// TIA Portal V17 export
// export: Created 2024-09-03T21:54:52.8265219Z, ExportSetting WithDefaults, DisplayName Totally Integrated Automation Portal, DisplayVersion V17 Update 7, DisplayName TIA Portal Openness, DisplayVersion V17 Update 7, DisplayName TIA Portal Version Control Interface, DisplayVersion V17, DisplayName SINAMICS Startdrive Advanced, DisplayVersion V17 SP2, DisplayName SINAMICS Startdrive G110M, G120, G120C, G120D, G120P, G115D, DisplayVersion V17 SP2, DisplayName SINAMICS Startdrive G130, G150, S120, S150, SINAMICS MV, S210, DisplayVersion V17 SP2, DisplayName STEP 7 Professional, DisplayVersion V17 Update 7, DisplayName STEP 7 Safety, DisplayVersion V17 Update 6, DisplayName WinCC Advanced / Unified PC, DisplayVersion V17 Update 7
FUNCTION_BLOCK "FB_Eks"   // FB5050, LAD
{ S7_Optimized_Access := 'TRUE' }
VERSION : 0.1
// stored: AutoNumber false, IsIECCheckEnabled false, IsRetainMemResEnabled false, MemoryReserve 100, SetENOAutomatically false, UDAEnableTagReadback false
   VAR_INPUT
      iScreenNumberEqual : Bool;
      iOpSwitchManualMode : Bool;
      iGenerateTimeoutError : Bool;
      iPermanentAccess : Bool;
      iBlinker : Bool;
   END_VAR
   VAR_OUTPUT
      qManualModeActive : Bool;
      qOpManualModeLamp : Bool;
      qeKeyTimeout : Bool;
   END_VAR
   VAR DB_SPECIFIC
      Status : Struct
         Key : Struct
            Inserted : Bool;
            Found : Bool;
            Valid : Bool;
            ActualKeyStatus : Int;   // 0= Not inserted, ??= GAP leader, ??= Maintenance, ??= Engineer, 100= Not registered
            LastKeyStatus : Int;   // 0= Not used, ??= GAP leader, ??= Maintenance, ??= Engineer, 100= Not registered
         END_STRUCT;
         Global : Struct
            GapLeader : Bool;
            Maintenance : Bool;
            Engineer : Bool;
            MaintenanceOrEngineer : Bool;
            AnyValidKey : Bool;
         END_STRUCT;
         ManualMode : Struct
            GapLeader : Bool;
            Maintenance : Bool;
            Engineer : Bool;
            MaintenanceOrEngineer : Bool;
            AnyValidKey : Bool;
         END_STRUCT;
      END_STRUCT;
   END_VAR
   VAR
      Database : Struct
         Status : Struct
            ActualAndLastKeyEqual { ExternalAccessible := 'False'; ExternalVisible := 'False'; ExternalWritable := 'False'} : Bool;
            LastKeyIsEmpty : Bool;
            LastKeyEmployeeIDIsEmpty : Bool;
            LastKeyFound { ExternalAccessible := 'False'; ExternalVisible := 'False'; ExternalWritable := 'False'} : Bool;
            LastKeyIndex { ExternalAccessible := 'False'; ExternalVisible := 'False'; ExternalWritable := 'False'} : Int;
            FreePlaceFound { ExternalAccessible := 'False'; ExternalVisible := 'False'; ExternalWritable := 'False'} : Bool;
            FreePlaceIndex { ExternalAccessible := 'False'; ExternalVisible := 'False'; ExternalWritable := 'False'} : Int;
            NumberOfKeys : Int;
            NumberOfStoredKeys : Int;
            StoredKeysReachedMaximum : Bool;
            NumberOfEngineerKeys : Int;
            NumberOfStoredEngineerKeys : Int;
            StoredEngineerKeysReachedMaximum : Bool;
         END_STRUCT;
         ListNumber : Int;
         ListNumberLast : Int;
      END_STRUCT;
   END_VAR
   VAR DB_SPECIFIC
      KeyManage : Struct
         CanBeAdd : Bool;
         Add : Bool;
         CanBeRemoved : Bool;
         Remove : Bool;
         CanBeUsed : Bool;
         Use : Int;
         CanBeSearched : Bool;
         Search : Bool;
         Searching : Bool;
         SearchedRow : Int;
         SearchedRowHMI : Int;
      END_STRUCT;
   END_VAR
   VAR RETAIN
      KeyTimeout : Time := T#2H_46M_39S;
   END_VAR
   VAR
      KeyInsertedInReader { S7_SetPoint := 'True'} : R_TRIG;
      KeyRemovedFromReader { S7_SetPoint := 'True'} : F_TRIG;
   END_VAR
   VAR DB_SPECIFIC
      TONs : Struct
         tDelayTimeoutError { S7_SetPoint := 'True'} : TON_TIME;
      END_STRUCT;
   END_VAR
   VAR_TEMP
      i : Int;
      stored_keys : Int;
      stored_engineer_keys : Int;
   END_VAR
   VAR_TEMP   // added for the SCL form of the ladder/FBD networks
      _w1 : Bool;
   END_VAR
BEGIN

REGION Network 1 (SCL): Inserted key
   //Key is inserted in reader
   #KeyInsertedInReader(CLK := "iEksKeyInserted");

   IF #KeyInsertedInReader.Q THEN
       "DB_EksData".LoadedData := "DB_EksData".EmptyKey;
       "DB_EksData".ActualKey := "DB_EksData".EmptyKey;
       #Status.Key.Inserted := TRUE;

       //Load level
       "DB_EksData".LoadedData.Level := "iEksLevel";

       //Load employee ID 
       "DB_EksData".LoadedData.EmployeeID[1] := "iEksEmployeeID_1";
       "DB_EksData".LoadedData.EmployeeID[2] := "iEksEmployeeID_2";
       "DB_EksData".LoadedData.EmployeeID[3] := "iEksEmployeeID_3";
       "DB_EksData".LoadedData.EmployeeID[4] := "iEksEmployeeID_4";

       //Adjust employee ID to be sure, that comparing with empty data will be coorect
       FOR #i := 1 TO 4 DO
           IF "DB_EksData".LoadedData.EmployeeID[#i] = '$00' THEN
               "DB_EksData".LoadedData.EmployeeID[#i] := ' ';
           END_IF;
       END_FOR;

       //Load key ID
       "FC_ByteToCharacters"(iByte := "iEksKeyID_1",
                             qChar1 => "DB_EksData".LoadedData.KeyID[1],
                             qChar2 => "DB_EksData".LoadedData.KeyID[2]);
       "FC_ByteToCharacters"(iByte := "iEksKeyID_2",
                             qChar1 => "DB_EksData".LoadedData.KeyID[3],
                             qChar2 => "DB_EksData".LoadedData.KeyID[4]);
       "FC_ByteToCharacters"(iByte := "iEksKeyID_3",
                             qChar1 => "DB_EksData".LoadedData.KeyID[5],
                             qChar2 => "DB_EksData".LoadedData.KeyID[6]);
       "FC_ByteToCharacters"(iByte := "iEksKeyID_4",
                             qChar1 => "DB_EksData".LoadedData.KeyID[7],
                             qChar2 => "DB_EksData".LoadedData.KeyID[8]);
       "FC_ByteToCharacters"(iByte := "iEksKeyID_5",
                             qChar1 => "DB_EksData".LoadedData.KeyID[9],
                             qChar2 => "DB_EksData".LoadedData.KeyID[10]);
       "FC_ByteToCharacters"(iByte := "iEksKeyID_6",
                             qChar1 => "DB_EksData".LoadedData.KeyID[11],
                             qChar2 => "DB_EksData".LoadedData.KeyID[12]);
       "FC_ByteToCharacters"(iByte := "iEksKeyID_7",
                             qChar1 => "DB_EksData".LoadedData.KeyID[13],
                             qChar2 => "DB_EksData".LoadedData.KeyID[14]);
       "FC_ByteToCharacters"(iByte := "iEksKeyID_8",
                             qChar1 => "DB_EksData".LoadedData.KeyID[15],
                             qChar2 => "DB_EksData".LoadedData.KeyID[16]);

       //Search inserted key in database
       FOR #i := 1 TO "EksNumberOfKeys" DO
           IF "DB_EksData".LoadedData.KeyID = "DB_EksList".Key[#i].KeyID THEN
               "DB_EksData".ActualKey := "DB_EksList".Key[#i];
               #Status.Key.Found := TRUE;
               IF "DB_EksList".Key[#i].Level = "EksGapLeaderLevel" OR
                   "DB_EksList".Key[#i].Level = "EksMaintenanceLevel" OR
                   "DB_EksList".Key[#i].Level = "EksEngineerLevel" THEN
                   #Status.Key.Valid := TRUE;
               END_IF;
               EXIT;
           END_IF;
       END_FOR;
       IF NOT #Status.Key.Found THEN
           "DB_EksData".ActualKey := "DB_EksData".LoadedData;
       END_IF;
   END_IF;

   //Key is removed from reader
   #KeyRemovedFromReader(CLK:="iEksKeyInserted");

   IF #KeyRemovedFromReader.Q THEN
       "DB_EksData".LastKey := "DB_EksData".ActualKey;
       "DB_EksData".ActualKey := "DB_EksData".EmptyKey;
   END_IF;

   //Manage data when key is not in reader or timeout error
   IF NOT "iEksKeyInserted" OR #qeKeyTimeout THEN
       #Status.Key.Inserted := FALSE;
       #Status.Key.Found := FALSE;
       #Status.Key.Valid := FALSE;
       #Status.Key.ActualKeyStatus := 0;
       "DB_EksData".ActualKey := "DB_EksData".EmptyKey;
   END_IF;

   //Reset timeout error
   IF NOT "iEksKeyInserted" THEN
       #qeKeyTimeout := FALSE;
   END_IF;
END_REGION

REGION Network 2: Set key status
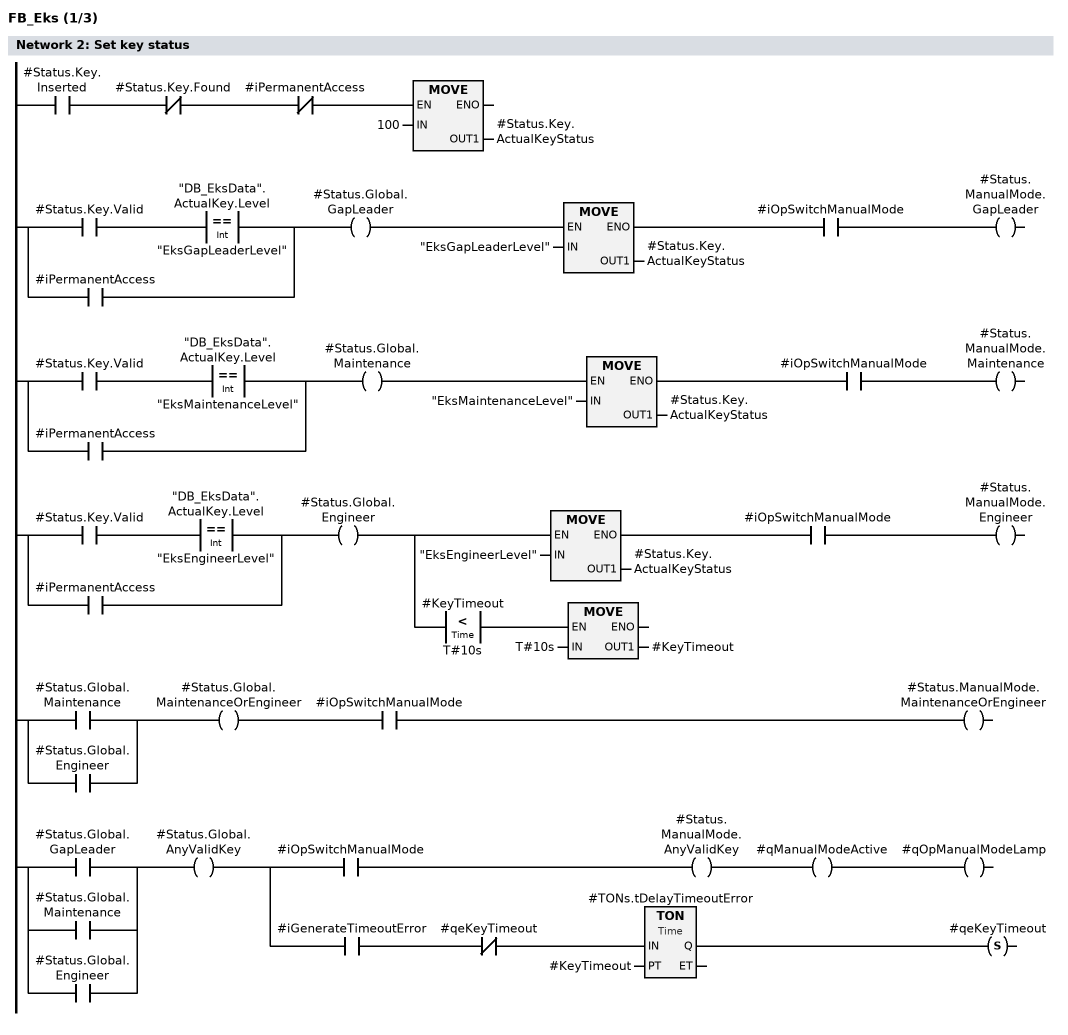
   RUNG wire#powerrail
      Contact( #Status.Key.Inserted )
      I_Contact( #Status.Key.Found )
      I_Contact( #iPermanentAccess )
      Move(in := 100, out1 => #Status.Key.ActualKeyStatus)
   END_RUNG
   RUNG wire#powerrail
      Contact( #Status.Key.Valid )
      { S7_Templates := "SrcType := Int" } EQ_Contact(in1 := "DB_EksData".ActualKey.Level, in2 := "EksGapLeaderLevel")
      wire#w1
      Coil( #Status.Global.GapLeader )
      Move(in := "EksGapLeaderLevel", out1 => #Status.Key.ActualKeyStatus)
      Contact( #iOpSwitchManualMode )
      Coil( #Status.ManualMode.GapLeader )
   END_RUNG
   RUNG wire#powerrail
      Contact( #iPermanentAccess )
   END_RUNG wire#w1
   RUNG wire#powerrail
      Contact( #Status.Key.Valid )
      { S7_Templates := "SrcType := Int" } EQ_Contact(in1 := "DB_EksData".ActualKey.Level, in2 := "EksMaintenanceLevel")
      wire#w2
      Coil( #Status.Global.Maintenance )
      Move(in := "EksMaintenanceLevel", out1 => #Status.Key.ActualKeyStatus)
      Contact( #iOpSwitchManualMode )
      Coil( #Status.ManualMode.Maintenance )
   END_RUNG
   RUNG wire#powerrail
      Contact( #iPermanentAccess )
   END_RUNG wire#w2
   RUNG wire#powerrail
      Contact( #Status.Key.Valid )
      { S7_Templates := "SrcType := Int" } EQ_Contact(in1 := "DB_EksData".ActualKey.Level, in2 := "EksEngineerLevel")
      wire#w3
      Coil( #Status.Global.Engineer )
      wire#w4
      Move(in := "EksEngineerLevel", out1 => #Status.Key.ActualKeyStatus)
      Contact( #iOpSwitchManualMode )
      Coil( #Status.ManualMode.Engineer )
   END_RUNG
   RUNG wire#powerrail
      Contact( #iPermanentAccess )
   END_RUNG wire#w3
   RUNG wire#w4
      { S7_Templates := "SrcType := Time" } LT_Contact(in1 := #KeyTimeout, in2 := T#10s)
      Move(in := T#10s, out1 => #KeyTimeout)
   END_RUNG
   RUNG wire#powerrail
      Contact( #Status.Global.Maintenance )
      wire#w5
      Coil( #Status.Global.MaintenanceOrEngineer )
      Contact( #iOpSwitchManualMode )
      Coil( #Status.ManualMode.MaintenanceOrEngineer )
   END_RUNG
   RUNG wire#powerrail
      Contact( #Status.Global.Engineer )
   END_RUNG wire#w5
   RUNG wire#powerrail
      Contact( #Status.Global.GapLeader )
      wire#w6
      Coil( #Status.Global.AnyValidKey )
      wire#w7
      Contact( #iOpSwitchManualMode )
      Coil( #Status.ManualMode.AnyValidKey )
      Coil( #qManualModeActive )
      Coil( #qOpManualModeLamp )
   END_RUNG
   RUNG wire#powerrail
      Contact( #Status.Global.Maintenance )
   END_RUNG wire#w6
   RUNG wire#powerrail
      Contact( #Status.Global.Engineer )
   END_RUNG wire#w6
   RUNG wire#w7
      Contact( #iGenerateTimeoutError )
      I_Contact( #qeKeyTimeout )
      { S7_Templates := "time_type := Time" } #TONs.tDelayTimeoutError.TON(pt := #KeyTimeout, et =>)
      S_Coil( #qeKeyTimeout )
   END_RUNG
   // the same network as SCL:
   IF #Status.Key.Inserted AND NOT #Status.Key.Found AND NOT #iPermanentAccess THEN
       #Status.Key.ActualKeyStatus := 100;
   END_IF;
   #Status.Global.GapLeader := (#Status.Key.Valid AND ("DB_EksData".ActualKey.Level = "EksGapLeaderLevel")) OR #iPermanentAccess;
   IF #Status.Global.GapLeader THEN #Status.Key.ActualKeyStatus := "EksGapLeaderLevel"; END_IF;
   #Status.ManualMode.GapLeader := #Status.Global.GapLeader AND #iOpSwitchManualMode;
   #Status.Global.Maintenance := (#Status.Key.Valid AND ("DB_EksData".ActualKey.Level = "EksMaintenanceLevel")) OR #iPermanentAccess;
   IF #Status.Global.Maintenance THEN #Status.Key.ActualKeyStatus := "EksMaintenanceLevel"; END_IF;
   #Status.ManualMode.Maintenance := #Status.Global.Maintenance AND #iOpSwitchManualMode;
   #Status.Global.Engineer := (#Status.Key.Valid AND ("DB_EksData".ActualKey.Level = "EksEngineerLevel")) OR #iPermanentAccess;
   IF #Status.Global.Engineer THEN #Status.Key.ActualKeyStatus := "EksEngineerLevel"; END_IF;
   #Status.ManualMode.Engineer := #Status.Global.Engineer AND #iOpSwitchManualMode;
   IF #Status.Global.Engineer AND (#KeyTimeout < T#10s) THEN #KeyTimeout := T#10s; END_IF;
   #Status.Global.MaintenanceOrEngineer := #Status.Global.Maintenance OR #Status.Global.Engineer;
   #Status.ManualMode.MaintenanceOrEngineer := #Status.Global.MaintenanceOrEngineer AND #iOpSwitchManualMode;
   #Status.Global.AnyValidKey := #Status.Global.GapLeader OR #Status.Global.Maintenance OR #Status.Global.Engineer;
   #Status.ManualMode.AnyValidKey := #Status.Global.AnyValidKey AND #iOpSwitchManualMode;
   #qManualModeActive := #Status.ManualMode.AnyValidKey;
   #qOpManualModeLamp := #Status.ManualMode.AnyValidKey;
   #TONs.tDelayTimeoutError.TON(IN := #Status.Global.AnyValidKey AND #iGenerateTimeoutError AND NOT #qeKeyTimeout,
                           PT := #KeyTimeout);
   IF #TONs.tDelayTimeoutError.Q THEN #qeKeyTimeout := TRUE; END_IF;
END_REGION

REGION Network 3 (SCL): Database status
   //Database status
   IF #iScreenNumberEqual THEN

       //Reset database status
       #Database.Status.ActualAndLastKeyEqual := FALSE;
       #Database.Status.LastKeyIsEmpty := FALSE;
       #Database.Status.LastKeyEmployeeIDIsEmpty := FALSE;
       #Database.Status.LastKeyFound := FALSE;
       #Database.Status.LastKeyIndex := 0;
       #Database.Status.FreePlaceFound := FALSE;
       #Database.Status.FreePlaceIndex := 0;
       #stored_keys := 0;
       #stored_engineer_keys := 0;

       //Compare actual and last inserted key
       IF #Status.Key.Inserted AND "DB_EksData".ActualKey.KeyID = "DB_EksData".LastKey.KeyID THEN
           //"DB_EksData".ActualKey.EmployeeID <> "DB_EksData".EmptyKey.EmployeeID THEN
           #Database.Status.ActualAndLastKeyEqual := TRUE;
       END_IF;

       //Last key is empty
       IF "DB_EksData".LastKey = "DB_EksData".EmptyKey THEN
           #Database.Status.LastKeyIsEmpty := TRUE;
       END_IF;

       //Last key employee ID is empty
       IF "DB_EksData".LastKey.EmployeeID = "DB_EksData".EmptyKey.EmployeeID THEN
           #Database.Status.LastKeyEmployeeIDIsEmpty := TRUE;
       END_IF;

       //Search database
       FOR #i := 1 TO "EksNumberOfKeys" DO

           //Search last key in database
           IF NOT #Database.Status.LastKeyFound AND
               "DB_EksData".LastKey.KeyID = "DB_EksList".Key[#i].KeyID THEN
               #Database.Status.LastKeyFound := TRUE;
               #Database.Status.LastKeyIndex := #i;
               #Status.Key.LastKeyStatus := "DB_EksData".LastKey.Level;
           END_IF;

           //Search free place in database            
           IF NOT #Database.Status.FreePlaceFound AND "DB_EksList".Key[#i] = "DB_EksData".EmptyKey THEN
               #Database.Status.FreePlaceFound := TRUE;
               #Database.Status.FreePlaceIndex := #i;
           END_IF;

           //Count stored keys
           IF "DB_EksList".Key[#i] <> "DB_EksData".EmptyKey THEN
               #stored_keys := #stored_keys + 1;

               IF "DB_EksList".Key[#i].Level = "EksEngineerLevel" THEN
                   #stored_engineer_keys := #stored_engineer_keys + 1;
               END_IF;

           END_IF;

       END_FOR;

       //Last key is not used
       IF #Database.Status.LastKeyIsEmpty THEN
           #Status.Key.LastKeyStatus := 0;
       END_IF;

       //Last key is not registered
       IF NOT #Database.Status.LastKeyIsEmpty AND NOT #Database.Status.LastKeyFound THEN
           #Status.Key.LastKeyStatus := 100;
       END_IF;

       //Check number of stored keys
       #Database.Status.NumberOfStoredKeys := #stored_keys;
       IF #Database.Status.NumberOfStoredKeys >= "EksNumberOfKeys" THEN
           #Database.Status.StoredKeysReachedMaximum := TRUE;
       ELSE
           #Database.Status.StoredKeysReachedMaximum := FALSE;
       END_IF;

       //Check number of stored engineer keys
       #Database.Status.NumberOfStoredEngineerKeys := #stored_engineer_keys;
       IF #Database.Status.NumberOfStoredEngineerKeys >= "EksNumberOfEngineerKeys" THEN
           #Database.Status.StoredEngineerKeysReachedMaximum := TRUE;
       ELSE
           #Database.Status.StoredEngineerKeysReachedMaximum := FALSE;
       END_IF;

   END_IF;
END_REGION

REGION Network 4: Add key
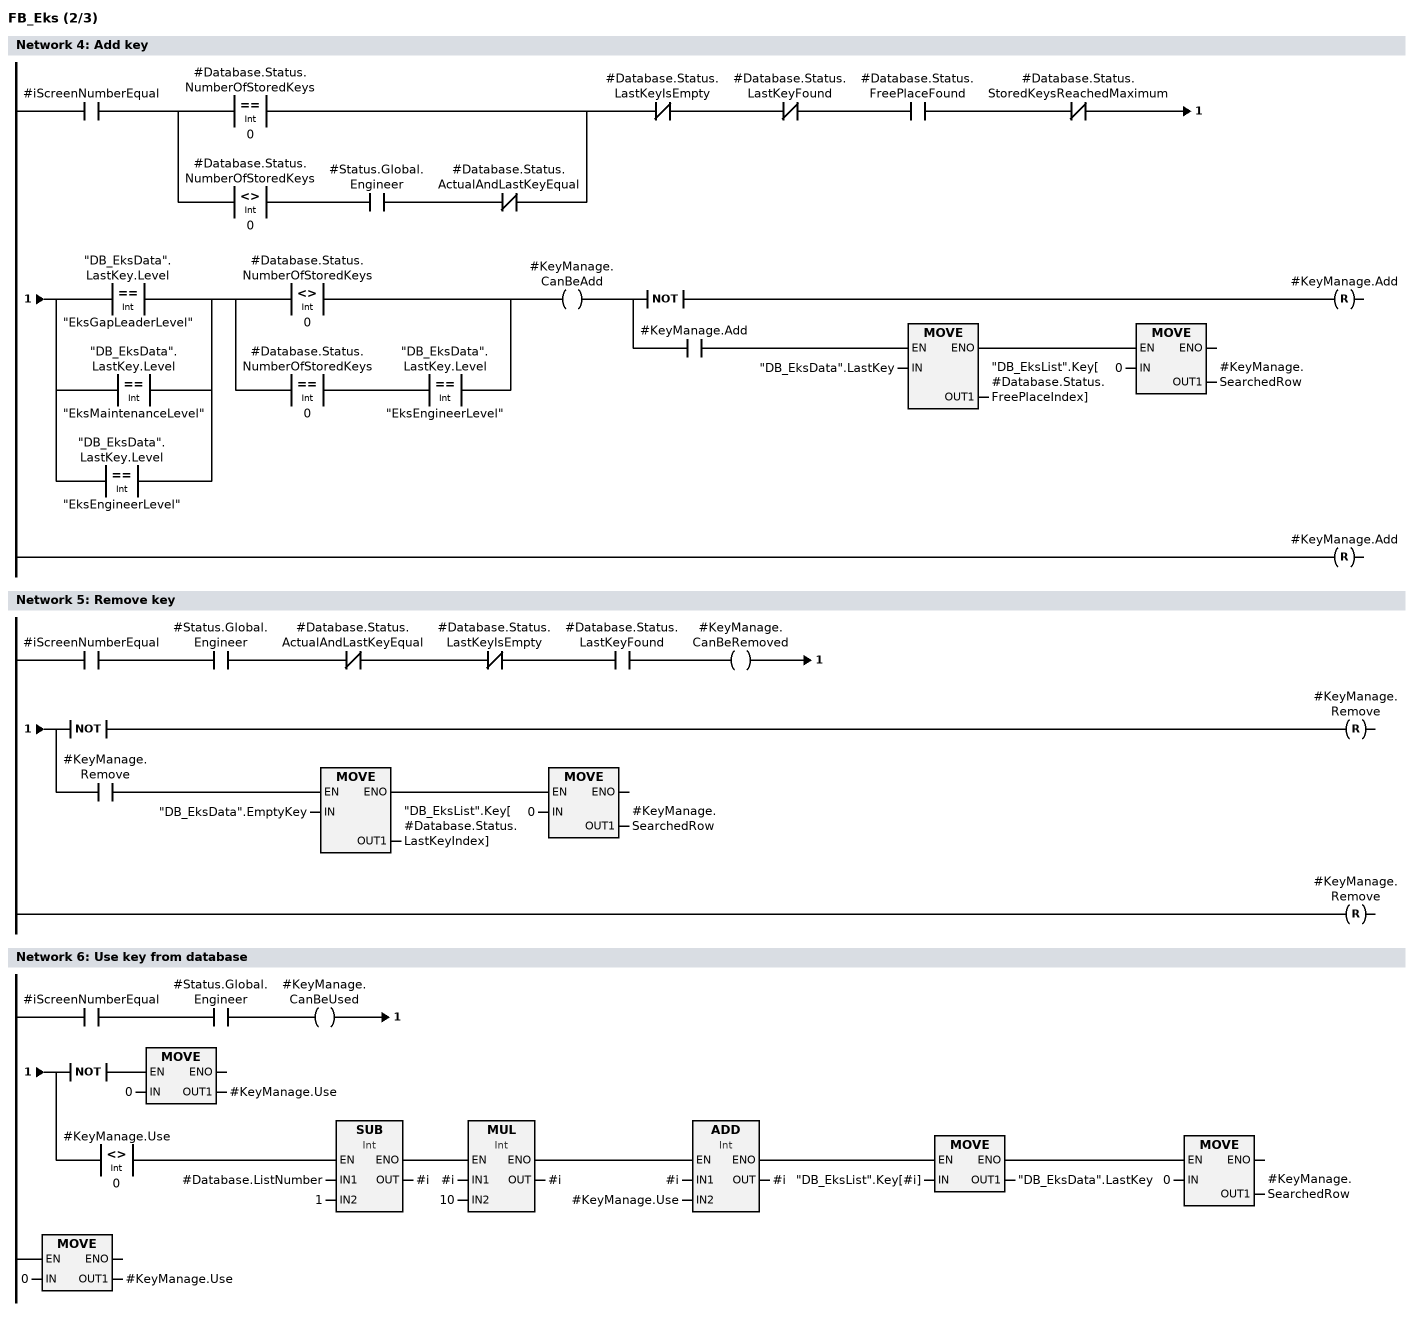
   RUNG wire#powerrail
      Contact( #iScreenNumberEqual )
      wire#w1
      { S7_Templates := "SrcType := Int" } EQ_Contact(in1 := #Database.Status.NumberOfStoredKeys, in2 := 0)
      wire#w2
      I_Contact( #Database.Status.LastKeyIsEmpty )
      I_Contact( #Database.Status.LastKeyFound )
      Contact( #Database.Status.FreePlaceFound )
      I_Contact( #Database.Status.StoredKeysReachedMaximum )
      wire#w3
      { S7_Templates := "SrcType := Int" } EQ_Contact(in1 := "DB_EksData".LastKey.Level, in2 := "EksGapLeaderLevel")
      wire#w4
      { S7_Templates := "SrcType := Int" } NE_Contact(in1 := #Database.Status.NumberOfStoredKeys, in2 := 0)
      wire#w5
      Coil( #KeyManage.CanBeAdd )
      wire#w6
      Not()
      R_Coil( #KeyManage.Add )
   END_RUNG
   RUNG wire#w1
      { S7_Templates := "SrcType := Int" } NE_Contact(in1 := #Database.Status.NumberOfStoredKeys, in2 := 0)
      Contact( #Status.Global.Engineer )
      I_Contact( #Database.Status.ActualAndLastKeyEqual )
   END_RUNG wire#w2
   RUNG wire#w3
      { S7_Templates := "SrcType := Int" } EQ_Contact(in1 := "DB_EksData".LastKey.Level, in2 := "EksMaintenanceLevel")
   END_RUNG wire#w4
   RUNG wire#w3
      { S7_Templates := "SrcType := Int" } EQ_Contact(in1 := "DB_EksData".LastKey.Level, in2 := "EksEngineerLevel")
   END_RUNG wire#w4
   RUNG wire#w4
      { S7_Templates := "SrcType := Int" } EQ_Contact(in1 := #Database.Status.NumberOfStoredKeys, in2 := 0)
      { S7_Templates := "SrcType := Int" } EQ_Contact(in1 := "DB_EksData".LastKey.Level, in2 := "EksEngineerLevel")
   END_RUNG wire#w5
   RUNG wire#w6
      Contact( #KeyManage.Add )
      Move(in := "DB_EksData".LastKey, out1 => "DB_EksList".Key[#Database.Status.FreePlaceIndex])
      Move(in := 0, out1 => #KeyManage.SearchedRow)
   END_RUNG
   RUNG wire#powerrail
      R_Coil( #KeyManage.Add )
   END_RUNG
   // the same network as SCL:
   #KeyManage.CanBeAdd := #iScreenNumberEqual AND ((#Database.Status.NumberOfStoredKeys = 0) OR ((#Database.Status.NumberOfStoredKeys <> 0) AND #Status.Global.Engineer AND NOT #Database.Status.ActualAndLastKeyEqual)) AND NOT #Database.Status.LastKeyIsEmpty AND NOT #Database.Status.LastKeyFound AND #Database.Status.FreePlaceFound AND NOT #Database.Status.StoredKeysReachedMaximum AND (("DB_EksData".LastKey.Level = "EksGapLeaderLevel") OR ("DB_EksData".LastKey.Level = "EksMaintenanceLevel") OR ("DB_EksData".LastKey.Level = "EksEngineerLevel")) AND ((#Database.Status.NumberOfStoredKeys <> 0) OR ((#Database.Status.NumberOfStoredKeys = 0) AND ("DB_EksData".LastKey.Level = "EksEngineerLevel")));
   IF NOT #KeyManage.CanBeAdd THEN #KeyManage.Add := FALSE; END_IF;
   IF #KeyManage.CanBeAdd AND #KeyManage.Add THEN
       "DB_EksList".Key[#Database.Status.FreePlaceIndex] := "DB_EksData".LastKey;
       #KeyManage.SearchedRow := 0;
   END_IF;
   #KeyManage.Add := FALSE;
END_REGION

REGION Network 5: Remove key
   RUNG wire#powerrail
      Contact( #iScreenNumberEqual )
      Contact( #Status.Global.Engineer )
      I_Contact( #Database.Status.ActualAndLastKeyEqual )
      I_Contact( #Database.Status.LastKeyIsEmpty )
      Contact( #Database.Status.LastKeyFound )
      Coil( #KeyManage.CanBeRemoved )
      wire#w1
      Not()
      R_Coil( #KeyManage.Remove )
   END_RUNG
   RUNG wire#w1
      Contact( #KeyManage.Remove )
      Move(in := "DB_EksData".EmptyKey, out1 => "DB_EksList".Key[#Database.Status.LastKeyIndex])
      Move(in := 0, out1 => #KeyManage.SearchedRow)
   END_RUNG
   RUNG wire#powerrail
      R_Coil( #KeyManage.Remove )
   END_RUNG
   // the same network as SCL:
   #KeyManage.CanBeRemoved := #iScreenNumberEqual AND #Status.Global.Engineer AND NOT #Database.Status.ActualAndLastKeyEqual AND NOT #Database.Status.LastKeyIsEmpty AND #Database.Status.LastKeyFound;
   IF NOT #KeyManage.CanBeRemoved THEN #KeyManage.Remove := FALSE; END_IF;
   IF #KeyManage.CanBeRemoved AND #KeyManage.Remove THEN
       "DB_EksList".Key[#Database.Status.LastKeyIndex] := "DB_EksData".EmptyKey;
       #KeyManage.SearchedRow := 0;
   END_IF;
   #KeyManage.Remove := FALSE;
END_REGION

REGION Network 6: Use key from database
   RUNG wire#powerrail
      Contact( #iScreenNumberEqual )
      Contact( #Status.Global.Engineer )
      Coil( #KeyManage.CanBeUsed )
      wire#w1
      Not()
      Move(in := 0, out1 => #KeyManage.Use)
   END_RUNG
   RUNG wire#w1
      { S7_Templates := "SrcType := Int" } NE_Contact(in1 := #KeyManage.Use, in2 := 0)
      { S7_Templates := "SrcType := Int" } Sub(in1 := #Database.ListNumber, in2 := 1, out => #i)
      { S7_Templates := "SrcType := Int" } Mul(in1 := #i, in2 := 10, out => #i)
      { S7_Templates := "SrcType := Int" } Add(in1 := #i, in2 := #KeyManage.Use, out => #i)
      Move(in := "DB_EksList".Key[#i], out1 => "DB_EksData".LastKey)
      Move(in := 0, out1 => #KeyManage.SearchedRow)
   END_RUNG
   RUNG wire#powerrail
      Move(in := 0, out1 => #KeyManage.Use)
   END_RUNG
   // the same network as SCL:
   #KeyManage.CanBeUsed := #iScreenNumberEqual AND #Status.Global.Engineer;
   IF NOT #KeyManage.CanBeUsed THEN #KeyManage.Use := 0; END_IF;
   IF #KeyManage.CanBeUsed AND (#KeyManage.Use <> 0) THEN
       #i := #Database.ListNumber - 1;
       #i := #i * 10;
       #i := #i + #KeyManage.Use;
       "DB_EksData".LastKey := "DB_EksList".Key[#i];
       #KeyManage.SearchedRow := 0;
   END_IF;
   #KeyManage.Use := 0;
END_REGION

REGION Network 7: Search last inserted key
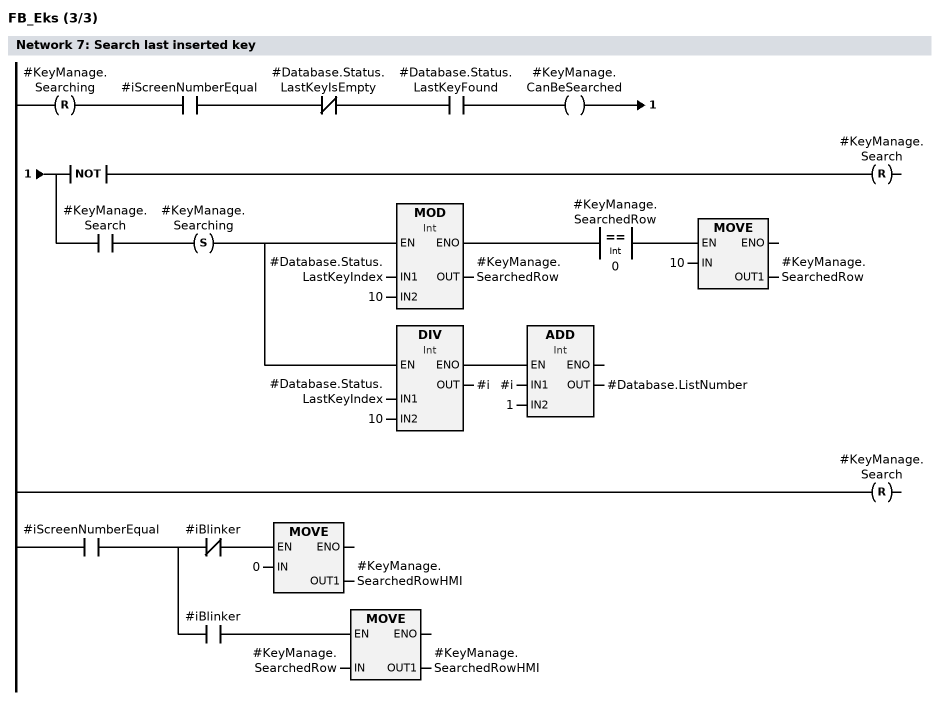
   RUNG wire#powerrail
      R_Coil( #KeyManage.Searching )
      Contact( #iScreenNumberEqual )
      I_Contact( #Database.Status.LastKeyIsEmpty )
      Contact( #Database.Status.LastKeyFound )
      Coil( #KeyManage.CanBeSearched )
      wire#w1
      Not()
      R_Coil( #KeyManage.Search )
   END_RUNG
   RUNG wire#w1
      Contact( #KeyManage.Search )
      S_Coil( #KeyManage.Searching )
      wire#w2
      { S7_Templates := "SrcType := Int" } Mod(in1 := #Database.Status.LastKeyIndex, in2 := 10, out => #KeyManage.SearchedRow)
      { S7_Templates := "SrcType := Int" } EQ_Contact(in1 := #KeyManage.SearchedRow, in2 := 0)
      Move(in := 10, out1 => #KeyManage.SearchedRow)
   END_RUNG
   RUNG wire#w2
      { S7_Templates := "SrcType := Int" } Div(in1 := #Database.Status.LastKeyIndex, in2 := 10, out => #i)
      { S7_Templates := "SrcType := Int" } Add(in1 := #i, in2 := 1, out => #Database.ListNumber)
   END_RUNG
   RUNG wire#powerrail
      R_Coil( #KeyManage.Search )
   END_RUNG
   RUNG wire#powerrail
      Contact( #iScreenNumberEqual )
      wire#w3
      I_Contact( #iBlinker )
      Move(in := 0, out1 => #KeyManage.SearchedRowHMI)
   END_RUNG
   RUNG wire#w3
      Contact( #iBlinker )
      Move(in := #KeyManage.SearchedRow, out1 => #KeyManage.SearchedRowHMI)
   END_RUNG
   // the same network as SCL:
   #KeyManage.Searching := FALSE;
   #KeyManage.CanBeSearched := #iScreenNumberEqual AND NOT #Database.Status.LastKeyIsEmpty AND #Database.Status.LastKeyFound;
   IF NOT #KeyManage.CanBeSearched THEN #KeyManage.Search := FALSE; END_IF;
   #_w1 := #KeyManage.CanBeSearched AND #KeyManage.Search;
   IF #_w1 THEN
       #KeyManage.Searching := TRUE;
       #KeyManage.SearchedRow := #Database.Status.LastKeyIndex MOD 10;
   END_IF;
   IF #_w1 AND (#KeyManage.SearchedRow = 0) THEN #KeyManage.SearchedRow := 10; END_IF;
   IF #_w1 THEN
       #i := #Database.Status.LastKeyIndex / 10;
       #Database.ListNumber := #i + 1;
   END_IF;
   #KeyManage.Search := FALSE;
   IF #iScreenNumberEqual AND NOT #iBlinker THEN #KeyManage.SearchedRowHMI := 0; END_IF;
   IF #iScreenNumberEqual AND #iBlinker THEN #KeyManage.SearchedRowHMI := #KeyManage.SearchedRow; END_IF;
END_REGION

REGION Network 8 (SCL): Key listing
   //List number limits
   IF #Database.ListNumber < 1 THEN
       #Database.ListNumber := 1;
   END_IF;

   #i := "EksNumberOfKeys" / 10;
   IF #Database.ListNumber > #i THEN
       #Database.ListNumber := #i;
   END_IF;

   //Keys limit
   #Database.Status.NumberOfKeys := "EksNumberOfKeys";
   #Database.Status.NumberOfEngineerKeys := "EksNumberOfEngineerKeys";

   //Reset searched row
   IF NOT #iScreenNumberEqual THEN
       #KeyManage.SearchedRow := 0;
   END_IF;

   IF #Database.ListNumberLast <> #Database.ListNumber THEN
       #Database.ListNumberLast := #Database.ListNumber;

       IF NOT #KeyManage.Searching THEN
           #KeyManage.SearchedRow := 0;
       END_IF;

   END_IF;

   //Key listing
   IF #iScreenNumberEqual THEN
       #i := (#Database.ListNumber - 1) * 10;
       "DB_EksData".KeyListHMI[1] := "DB_EksList".Key[#i + 1];
       "DB_EksData".KeyListHMI[2] := "DB_EksList".Key[#i + 2];
       "DB_EksData".KeyListHMI[3] := "DB_EksList".Key[#i + 3];
       "DB_EksData".KeyListHMI[4] := "DB_EksList".Key[#i + 4];
       "DB_EksData".KeyListHMI[5] := "DB_EksList".Key[#i + 5];
       "DB_EksData".KeyListHMI[6] := "DB_EksList".Key[#i + 6];
       "DB_EksData".KeyListHMI[7] := "DB_EksList".Key[#i + 7];
       "DB_EksData".KeyListHMI[8] := "DB_EksList".Key[#i + 8];
       "DB_EksData".KeyListHMI[9] := "DB_EksList".Key[#i + 9];
       "DB_EksData".KeyListHMI[10] := "DB_EksList".Key[#i + 10];
   END_IF;
END_REGION
END_FUNCTION_BLOCK
